FUNCTION_BLOCK CoE_property_bool EXTENDS CoE_property
VAR_INPUT
END_VAR
VAR_OUTPUT
END_VAR
VAR
	_value : BOOL;
END_VAR

PROPERTY dataTypeSize : UINT
GET
dataTypeSize := SIZEOF(_value);
END_GET
END_PROPERTY

METHOD get_value : BOOL
VAR_OUTPUT
	value : bool ;
	errId : UDINT;
END_VAR
IF init_done THEN
	value := _value;
	get_value := TRUE;
ELSE
	errId := 2;
	get_value := FALSE;
END_IF
END_METHOD

METHOD handle_read_callback : BOOL
VAR_INPUT
	pt_buffer : POINTER TO CoE_buffer_type_cast_union;
	errId : UDINT;
END_VAR

_value := pt_buffer^.value_bool;
_init_done:=TRUE;
_read_errId:=errId;
END_METHOD

METHOD set_value : BOOL
VAR_INPUT
	value : bool ;
END_VAR
_valueToWrite.value_bool := value;
IF THIS^._I_CoE_communication_handler <> 0 THEN 
	THIS^._I_CoE_communication_handler.add_write_request(THIS^);
ELSE
	errId:=1;
END_IF
END_METHOD

END_FUNCTION_BLOCK

(* stored: Version 1.1.0.1, ProductVersion 3.1.4024.6
   POU CoE_property_bool: Id {c280b208-b524-007b-1e42-cbff16a2b75f}, SpecialFunc None
   Property dataTypeSize: Id {c0c533bd-17ea-0fee-154f-2bbbeb1b2849}
   Get Get: Id {0c4352cf-e01c-0a69-16cd-a741c9964472}
   Method get_value: Id {ef8435be-f0e5-078f-0cfa-f7a27d54ebcd}
   Method handle_read_callback: Id {25a981c3-4df0-0719-31e4-4422431b30db}
   Method set_value: Id {9a670921-a95b-03bc-1f30-83e9ec28fe9f} *)
